FUNCTION_BLOCK T_GetLastMsgLogger IMPLEMENTS I_Logger

VAR_OUTPUT
	lastLog : STRING;
	lasLogLevel : DWORD;
END_VAR

METHOD ToLog
VAR_INPUT
	Msg	: STRING(255);
	(* generic level, can be mapped to logging framework*)
	LogLevel	: DWORD;
END_VAR
lastLog := MSg;
lasLogLevel := LogLevel;
END_METHOD

END_FUNCTION_BLOCK

(* stored: Version 1.1.0.1, ProductVersion 3.1.4024.9
   POU T_GetLastMsgLogger: Id {cc23bc20-01af-46bf-8f0e-6dd882c31443}, SpecialFunc None
   Method ToLog: Id {e1ac84b0-4f69-4a30-a79b-953ef2b1eeab} *)
